// Factoryio modbus mapping for analog outputs
TYPE ST_ModbusMapHoldingRegs:
STRUCT
    // Gewicht
    nDispWeight: WORD;
    // Left count
    nDispCountLeft: WORD;
    // Forward count
    nDispCountForward: WORD;
    // Right count
    nDispCountRight: WORD;
    // nOut4
    {attribute 'hide'}
    nOut4: WORD;
    // FACTORY I/O (Camera Position)
    nFactoryCameraPosition: WORD;
END_STRUCT
END_TYPE

(* stored: Version 1.1.0.1
   DUT ST_ModbusMapHoldingRegs: Id {cd84abd8-76ae-43b6-9982-68711ffbfbd2} *)
